{attribute 'linkalways'} 
{attribute 'no_explicit_call' := 'This FB is a CLASS and must be accessed using methods or properties'}
{attribute 'enable_dynamic_creation'}
FUNCTION_BLOCK FINAL BooleanLiteralNode EXTENDS Node
VAR
	value : _BOOL(FALSE);
	out : _BOOL(FALSE);
END_VAR

METHOD PUBLIC Clone : I_Node
VAR
	pNode : POINTER TO BooleanLiteralNode;
END_VAR
pNode := __NEW(BooleanLiteralNode);
Clone := pNode^;
END_METHOD

METHOD FB_init : BOOL
VAR_INPUT
	bInitRetains : BOOL; // if TRUE, the retain variables are initialized (warm start / cold start)
	bInCopyCode : BOOL;  // if TRUE, the instance afterwards gets moved into the copy code (online change)
END_VAR
AddParameter('value', value);
AddOutput('out', out);
END_METHOD

METHOD PROTECTED OnExecute : HRESULT
VAR
END_VAR
out.value := value.value;
END_METHOD

END_FUNCTION_BLOCK

(* stored: Version 1.1.0.1, ProductVersion 3.1.4024.12
   POU BooleanLiteralNode: Id {d5e9096f-3db3-080c-2d3e-202427ce0cfa}, SpecialFunc None
   Folder Constructor: Id {c18534b5-81fd-4c4c-b7e1-6df55c1d7b73}
   Method Clone: Id {eebef87a-b455-4952-a344-8e712682dbfa}
   Method FB_init: Id {ec68ff21-af02-414e-9b21-1672fdae5651}
   Method OnExecute: Id {d0655c70-f1d3-071d-3338-3d7948300785} *)
